// TIA Portal V19 export
TYPE "LEXCHANGETRAY_typeNgStrapInterface"
TITLE = exchangeTray_typeNgStrapInterface
// exchangeTray_typeNgStrapInterface related values
// stored: Access Published
   STRUCT
      configuration { ExternalAccessible := 'False'; ExternalVisible := 'False'; ExternalWritable := 'False'} : "LEXCHANGETRAY_typeNgStrapConfigeration";
      commands { ExternalAccessible := 'False'; ExternalVisible := 'False'; ExternalWritable := 'False'} : "LEXCHANGETRAY_typeNgStrapManualCommands";   // Module related manual commands from HMI
      monitoring { ExternalAccessible := 'False'; ExternalVisible := 'False'; ExternalWritable := 'False'} : "LEXCHANGETRAY_typeNgStrapProcessValues";
   END_STRUCT;
END_TYPE
